{attribute addProperty BoxType "EP7402-0057-0017"}
{attribute addProperty Id "OutputAT %Q*ARRAY[0 ..3] OF BOOL3240Control_outputAT %Q*ARRAY[0 ..3] OF BOOL3240"}
{attribute addProperty CRC "636064057"}
{attribute addProperty SizeInBites "64"}
{attribute addProperty SizeInBytes "8"}
TYPE DO_Outputs_43F80E28 :
STRUCT
	{attribute addProperty Name "Output"}
	Output AT %Q* : ARRAY[0 ..3] OF BOOL;
	{attribute addProperty Name "Control_output"}
	Control_output AT %Q* : ARRAY[0 ..3] OF BOOL;
END_STRUCT
END_TYPE

(* stored: Version 1.2.0.0, ProductVersion 3.1.4024.9
   DUT DO_Outputs_43F80E28: Id {b5d48879-069b-4b72-bfb9-e7d70acddfba} *)
